// TIA Portal project "Motor_Paso_Paso" (V17)

(* hardware
DEVICE "S7-1200 station_1"  S7-1200 Station
   slot 0: "Rack_0"  S7-1200 Rack  Rack  V1.0
   slot 1: "PLC_1"  CPU 1214C DC/DC/DC  6ES7 214-1AG40-0XB0  V4.3
   slot 2: "DI 8x24VDC_1"  6ES7 221-1BF32-0XB0  V2.0
*)

// ===== PLC "PLC_1"  CPU 1214C DC/DC/DC =====

VAR_GLOBAL   // PLC tag table "Default tag table"
   "Clock_Byte" AT %MB0 : Byte;
   "Clock_10Hz" AT %M0.0 : Bool;
   "Clock_5Hz" AT %M0.1 : Bool;
   "Clock_2.5Hz" AT %M0.2 : Bool;
   "Clock_2Hz" AT %M0.3 : Bool;
   "Clock_1.25Hz" AT %M0.4 : Bool;
   "Clock_1Hz" AT %M0.5 : Bool;
   "Clock_0.625Hz" AT %M0.6 : Bool;
   "Clock_0.5Hz" AT %M0.7 : Bool;
   "System_Byte" AT %MB1 : Byte;
   "FirstScan" AT %M1.0 : Bool;
   "DiagStatusUpdate" AT %M1.1 : Bool;
   "AlwaysTRUE" AT %M1.2 : Bool;
   "AlwaysFALSE" AT %M1.3 : Bool;
   "IA00" AT %I0.0 : Bool;
   "IA01" AT %I0.1 : Bool;
   "IA02" AT %I0.2 : Bool;
   "IA03" AT %I0.3 : Bool;
   "IA04" AT %I0.4 : Bool;
   "IA05" AT %I0.5 : Bool;
   "IA06" AT %I0.6 : Bool;
   "IA07" AT %I0.7 : Bool;
   "IB00" AT %I1.0 : Bool;
   "IB01" AT %I1.1 : Bool;
   "IB02" AT %I1.2 : Bool;
   "IB03" AT %I1.3 : Bool;
   "IB04" AT %I1.4 : Bool;
   "IB05" AT %I1.5 : Bool;
   "IB06" AT %I1.6 : Bool;
   "IB07" AT %I1.7 : Bool;
   "QA00" AT %Q0.0 : Bool;
   "QA01" AT %Q0.1 : Bool;
   "QA02" AT %Q0.2 : Bool;
   "QA03" AT %Q0.3 : Bool;
   "QA04" AT %Q0.4 : Bool;
   "QA05" AT %Q0.5 : Bool;
   "QA06" AT %Q0.6 : Bool;
   "QA07" AT %Q0.7 : Bool;
   "QB00" AT %Q1.0 : Bool;
   "QB01" AT %Q1.1 : Bool;
   "QB02" AT %Q1.2 : Bool;
   "QB03" AT %Q1.3 : Bool;
   "QB04" AT %Q1.4 : Bool;
   "QB05" AT %Q1.5 : Bool;
   "QB06" AT %Q1.6 : Bool;
   "QB07" AT %Q1.7 : Bool;
   "Axis_X_Enable" AT %M100.0 : Bool;
   "Axis_X_CW_Ready" AT %M100.1 : Bool;
   "Axis_X_Sensor_Homming" AT %M100.2 : Bool;
   "Axis_X_CCW_Ready" AT %M100.3 : Bool;
   "Axis_Y_Enable" AT %M200.0 : Bool;
   "Axis_Y_CW_Ready" AT %M200.1 : Bool;
   "Axis_Y_Sensor_Homming" AT %M200.2 : Bool;
   "Axis_Y_CCW_Ready" AT %M200.3 : Bool;
END_VAR

DATA_BLOCK "MD5-HD14"   // DB1
{ S7_Optimized_Access := 'TRUE' }
VERSION : 0.1
   VAR RETAIN
      Axis_X : Struct
         Start : Bool;
         Stop : Bool;
         Select_Direction : Bool;
         CW_Direction : Bool;
         CCW_Direction : Bool;
         Reset : Bool;
         Enable_Jog_Mov : Bool;
         Enable_Rel_Mov : Bool;
         Enable_Abs_Mov : Bool;
         Position_Abs : Real;
         Position_Rel : Real;
         Velocity : Real := 4.0;
         Axis_X : Struct
            Start : Bool;
            Stop : Bool;
            Select_Direction : Bool;
            CW_Direction : Bool;
            CCW_Direction : Bool;
            Reset : Bool;
            Enable : Bool;
            Position : Real;
            Velocity : Real;
         END_STRUCT;
      END_STRUCT;
      Axis_Y : Struct
         Start : Bool;
         Stop : Bool;
         Select_Direction : Bool;
         CW_Direction : Bool;
         CCW_Direction : Bool;
         Reset : Bool;
         Enable : Bool;
         Position : Real;
         Velocity : Real := 4.5;
         Axis_X : Struct
            Start : Bool;
            Stop : Bool;
            Select_Direction : Bool;
            CW_Direction : Bool;
            CCW_Direction : Bool;
            Reset : Bool;
            Enable : Bool;
            Position : Real;
            Velocity : Real;
         END_STRUCT;
      END_STRUCT;
   END_VAR
   VAR
      Aux_Pulses : Array[0..10] of Bool;
   END_VAR
BEGIN
END_DATA_BLOCK

DATA_BLOCK "General"   // DB3
{ S7_Optimized_Access := 'TRUE' }
VERSION : 0.1
   VAR
      In : Struct
         Emergency_Stop : Bool;
         Reset_Button : Bool;
         Bimanual_01 : Bool;
         Bimanual_02 : Bool;
         Presostate : Bool;
         Spare : Array[0..16] of Bool;
      END_STRUCT;
      Out : Struct
         Step_Motor_01_CW : Bool;
         Step_Motor_01_CCW : Bool;
         Step_Motor_02_CW : Bool;
         Step_Motor_02_CCW : Bool;
      END_STRUCT;
   END_VAR
BEGIN
END_DATA_BLOCK

DATA_BLOCK "Axis_X_CW_CCW"   // DB2, Motion_DB
{ S7_Optimized_Access := 'TRUE' }
AUTHOR : SIMATIC
FAMILY : BasicMC
NAME : TO_PosAx
VERSION : 6.0
// stored: InstanceOfName TO_PositioningAxis
"TO_PositioningAxis"
BEGIN
   // Axis.DirectionOutputEnabledCU = TRUE
   // Axis.LengthUnitNormalized.Distance = 1013
   // Axis.OnlinePtoModeCU = 16#0000_0003
   // Axis.SelectedChannel2EnumCU = %Q0.1
   // Axis.SelectedChannel1EnumCU = %Q0.0
   // Pulse.MinDeltaDeltaFrequencyCU = 0.004
   // Pulse.MaxDeltaDeltaFrequencyCU = 1.0E+10
   // Pulse.MinDeltaFrequencyCU = 0.005
   // Pulse.MaxDeltaFrequencyCU = 9.5E+9
   // Pulse.MinFrequencyCU = 1.0
   // Pulse.MaxFrequencyCU = 100000.0
   // Pulse.OutputSourceCU = 16#0000_0000
   // Axis.SelectPTO = 0
END_DATA_BLOCK

DATA_BLOCK "Axis_Y_CW_CCW"   // DB7, Motion_DB
{ S7_Optimized_Access := 'TRUE' }
AUTHOR : SIMATIC
FAMILY : BasicMC
NAME : TO_PosAx
VERSION : 6.0
// stored: InstanceOfName TO_PositioningAxis
"TO_PositioningAxis"
BEGIN
   // Axis.DirectionOutputEnabledCU = TRUE
   // Axis.LengthUnitNormalized.Distance = 1013
   // Axis.OnlinePtoModeCU = 16#0000_0002
   // Axis.SelectedChannel2EnumCU = %Q0.3
   // Axis.SelectedChannel1EnumCU = %Q0.2
   // Pulse.MinDeltaDeltaFrequencyCU = 0.004
   // Pulse.MaxDeltaDeltaFrequencyCU = 1.0E+10
   // Pulse.MinDeltaFrequencyCU = 0.005
   // Pulse.MaxDeltaFrequencyCU = 9.5E+9
   // Pulse.MinFrequencyCU = 1.0
   // Pulse.MaxFrequencyCU = 100000.0
   // Pulse.OutputSourceCU = 16#0000_0000
   // Axis.SelectPTO = 1
   // Axis.OnlinePtoIndexCU = 1
END_DATA_BLOCK

FUNCTION "A002- Assing IO's" : Void   // FC1, LAD
{ S7_Optimized_Access := 'TRUE' }
VERSION : 0.1
BEGIN

REGION Network 1 (SCL): Assing IA00 to IA07
   IF "AlwaysTRUE" THEN
       "General".In.Presostate     := "IA00";
       "General".In.Emergency_Stop := "IA01";
       "General".In.Bimanual_01    := "IA02";
       "General".In.Bimanual_02    := "IA03";
       "General".In.Spare[4]       := "IA04";
       "General".In.Spare[5]       := "IA05";
       "General".In.Spare[6]       := "IA06";
       "General".In.Spare[7]       := "IA07";


       "General".In.Spare[8]       := "IB00";
       "General".In.Spare[9]       := "IB01";
       "General".In.Spare[10]      := "IB02";
       "General".In.Spare[11]      := "IB03";
       "General".In.Spare[12]      := "IB04";
       "General".In.Spare[13]      := "IB05";
       "General".In.Spare[14]      := "IB06";
       "General".In.Spare[15]      := "IB07";
       ;
   END_IF;
END_REGION

REGION Network 2 (SCL): Assing QA00 to QA07
   //IF "AlwaysTRUE" THEN
   //    "QA00" := "General".Out.Step_Motor_01_CW;
   //    "QA01" := "General".Out.Step_Motor_01_CCW;
   //    "QA02" := "General".Out.Step_Motor_02_CW;
   //    "QA03" := "General".Out.Step_Motor_02_CCW;
   //    ;
   //END_IF;
END_REGION
END_FUNCTION

FUNCTION "A020- Motion Control MPP" : Void   // FC20, LAD
{ S7_Optimized_Access := 'TRUE' }
VERSION : 0.1
   VAR_TEMP   // added for the SCL form of the ladder/FBD networks
      _w1 : Bool;
   END_VAR
BEGIN

REGION Network 1: Enable MC Power of Motors
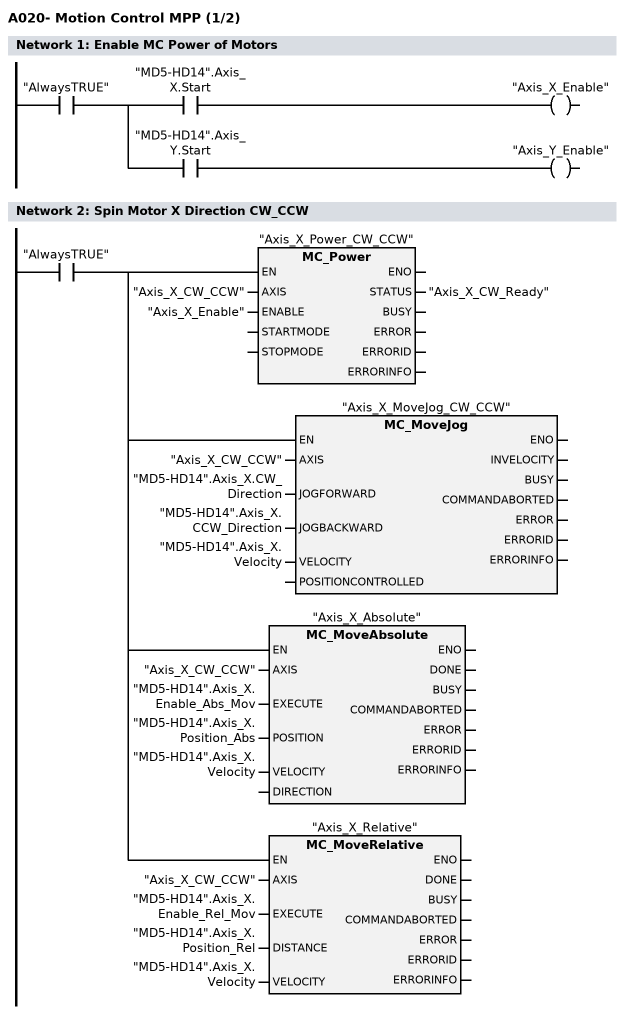
   RUNG wire#powerrail
      Contact( "AlwaysTRUE" )
      wire#w1
      Contact( "MD5-HD14".Axis_X.Start )
      Coil( "Axis_X_Enable" )
   END_RUNG
   RUNG wire#w1
      Contact( "MD5-HD14".Axis_Y.Start )
      Coil( "Axis_Y_Enable" )
   END_RUNG
   // the same network as SCL:
   "Axis_X_Enable" := "AlwaysTRUE" AND "MD5-HD14".Axis_X.Start;
   "Axis_Y_Enable" := "AlwaysTRUE" AND "MD5-HD14".Axis_Y.Start;
END_REGION

REGION Network 2: Spin Motor X Direction CW_CCW
   #_w1 := "AlwaysTRUE";
   IF #_w1 THEN
       "Axis_X_Power_CW_CCW"(Axis := "Axis_X_CW_CCW", Enable := "Axis_X_Enable", Status => "Axis_X_CW_Ready");   // MC_Power
       "Axis_X_MoveJog_CW_CCW"(Axis := "Axis_X_CW_CCW",   // MC_MoveJog
                               JogForward := "MD5-HD14".Axis_X.CW_Direction,
                               JogBackward := "MD5-HD14".Axis_X.CCW_Direction,
                               Velocity := "MD5-HD14".Axis_X.Velocity);
       "Axis_X_Absolute"(Axis := "Axis_X_CW_CCW",   // MC_MoveAbsolute
                         Execute := "MD5-HD14".Axis_X.Enable_Abs_Mov,
                         Position := "MD5-HD14".Axis_X.Position_Abs,
                         Velocity := "MD5-HD14".Axis_X.Velocity);
       "Axis_X_Relative"(Axis := "Axis_X_CW_CCW",   // MC_MoveRelative
                         Execute := "MD5-HD14".Axis_X.Enable_Rel_Mov,
                         Distance := "MD5-HD14".Axis_X.Position_Rel,
                         Velocity := "MD5-HD14".Axis_X.Velocity);
   END_IF;
END_REGION

REGION Network 3: Spin Motor Y Direction CW_CCW
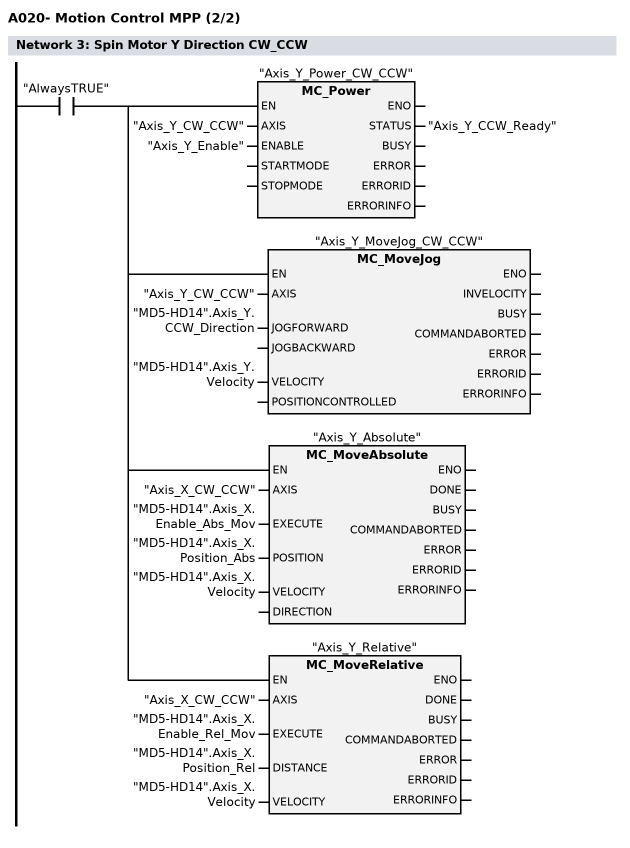
   #_w1 := "AlwaysTRUE";
   IF #_w1 THEN
       "Axis_Y_Power_CW_CCW"(Axis := "Axis_Y_CW_CCW", Enable := "Axis_Y_Enable", Status => "Axis_Y_CCW_Ready");   // MC_Power
       "Axis_Y_MoveJog_CW_CCW"(Axis := "Axis_Y_CW_CCW",   // MC_MoveJog
                               JogForward := "MD5-HD14".Axis_Y.CCW_Direction,
                               Velocity := "MD5-HD14".Axis_Y.Velocity);
       "Axis_Y_Absolute"(Axis := "Axis_X_CW_CCW",   // MC_MoveAbsolute
                         Execute := "MD5-HD14".Axis_X.Enable_Abs_Mov,
                         Position := "MD5-HD14".Axis_X.Position_Abs,
                         Velocity := "MD5-HD14".Axis_X.Velocity);
       "Axis_Y_Relative"(Axis := "Axis_X_CW_CCW",   // MC_MoveRelative
                         Execute := "MD5-HD14".Axis_X.Enable_Rel_Mov,
                         Distance := "MD5-HD14".Axis_X.Position_Rel,
                         Velocity := "MD5-HD14".Axis_X.Velocity);
   END_IF;
END_REGION
END_FUNCTION

ORGANIZATION_BLOCK "A001- Main"   // OB1, LAD, ProgramCycle
TITLE = "Main Program Sweep (Cycle)"
{ S7_Optimized_Access := 'TRUE' }
VERSION : 0.1
   VAR_INPUT
      Initial_Call : Bool;   // Initial call of this OB
      Remanence : Bool;   // =True, if remanent data are available
   END_VAR
BEGIN

REGION Network 1: Call Assing IO's
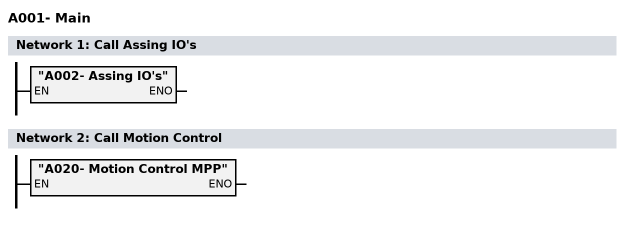
   RUNG wire#powerrail
      "A002- Assing IO's"()
   END_RUNG
   // the same network as SCL:
   "A002- Assing IO's"();
END_REGION

REGION Network 2: Call Motion Control
   RUNG wire#powerrail
      "A020- Motion Control MPP"()
   END_RUNG
   // the same network as SCL:
   "A020- Motion Control MPP"();
END_REGION
END_ORGANIZATION_BLOCK